// Implicitly generated code : DO NOT EDIT
FUNCTION CheckDivReal : REAL
VAR_INPUT
	divisor:REAL;
END_VAR

// Implicitly generated code : Only an Implementation suggestion
{noflow}
IF divisor = 0 THEN
	CheckDivReal:=1;
ELSE
	CheckDivReal:=divisor;
END_IF;
{flow}

END_FUNCTION

(* stored: Version 1.1.0.1, ProductVersion 3.1.4022.18
   POU CheckDivReal: Id {a2363707-0ca8-478a-ab80-f8e64d831dd5}, SpecialFunc CheckDivReal32 *)
